TYPE ST_Fanuc_ManPos :
STRUCT
	nPosX				:REAL;
	nPosY				:REAL;
	nPosR				:REAL;
END_STRUCT
END_TYPE

(* stored: Version 1.1.0.1, ProductVersion 3.1.4024.11
   DUT ST_Fanuc_ManPos: Id {bfbea4f1-1ed3-4c56-84ed-ce5ffba62222} *)
